Omron CX-Programmer project NewProject (CX-Programmer 9.03)

# PLC NewPLC1: CJ1M CPU11
I/O table (CPU CJ1M-CPU11): rack 0 slot 0 CJ1W-OC211

## Global symbols (name address type ; comment)
0.00 BOOL  ; Tombol OFF
0.01 BOOL  ; Tombol ON
0.02 BOOL  ; sensor 1
0.03 BOOL  ; photosensor 2
0.04 BOOL  ; photosensor 3
0.05 BOOL  ; photosensor 4
100.00 BOOL  ; Memory Tombol ON
100.01 BOOL  ; Memory photosensor 1
100.02 BOOL  ; Motor On
100.03 BOOL  ; memory photosensor 1
100.04 BOOL  ; memory photosensor 3
100.05 BOOL  ; memory photosensor 4
10.00 BOOL  ; Deteksi Barang Ada/Tidak
10.01 BOOL  ; Deteksi Barang Palsu
10.02 BOOL  ; Menyimpan input sensor 1
10.03 BOOL  ; Reset input sensor 1
T0004 BOOL  ; timer off motor

## Program NewProgram1 (cyclic task 0)

### Section Section1

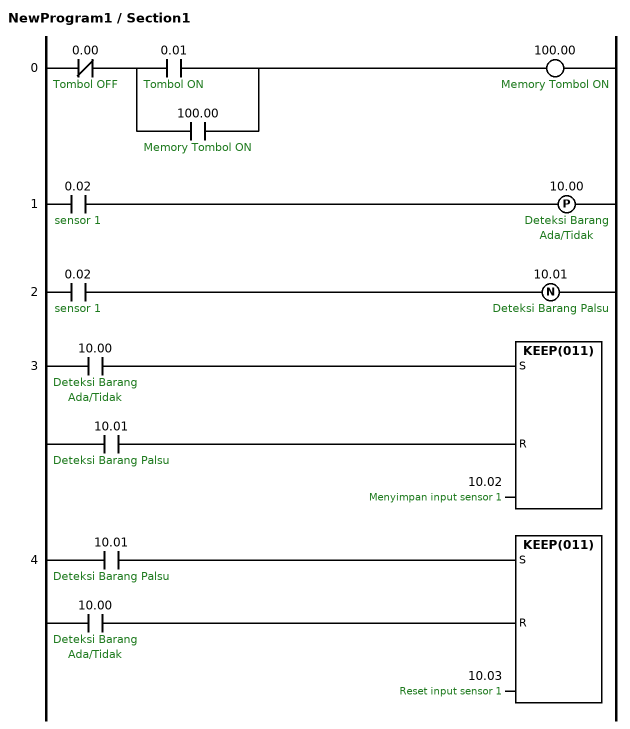
; rung 0
LDNOT 0.00  ; Tombol OFF
LD 0.01  ; Tombol ON
OR 100.00  ; Memory Tombol ON
ANDLD
OUT 100.00  ; Memory Tombol ON
; rung 1
LD 0.02  ; sensor 1
DIFU(013) 10.00  ; Deteksi Barang Ada/Tidak
; rung 2
LD 0.02  ; sensor 1
DIFD(014) 10.01  ; Deteksi Barang Palsu
; rung 3
LD 10.00  ; Deteksi Barang Ada/Tidak
LD 10.01  ; Deteksi Barang Palsu
KEEP(011) 10.02  ; Menyimpan input sensor 1
; rung 4
LD 10.01  ; Deteksi Barang Palsu
LD 10.00  ; Deteksi Barang Ada/Tidak
KEEP(011) 10.03  ; Reset input sensor 1

### Section END
; rung 0
END(001)